Omron CX-Programmer project Karosszeria_gyartosor (CX-Programmer 9.10)

# PLC PLC: CJ2M CPU32
I/O table (CPU CJ2M-CPU32): rack 0 slot 0 CJ1W-ID211; rack 0 slot 1 CJ1W-OD212; rack 0 slot 2 CJ1W-ID211; rack 0 slot 3 CJ1W-OD212; rack 0 slot 11 CJ2M-EIP21

## Global symbols (name address type ; comment)
CRANE_Seq_1 D90 UINT[10]  ; Az 1-es típusú karosszéria átemelési feladatának pozícióit tartalmazó tömb.
CRANE_Seq_1_Lenght D41 UINT  ; Az 1-es típusú karosszéria átemelési feladatának pozícióit tartalmazó tömb hossza.
CRANE_Seq_2 D107 UINT[8]  ; Az 2-es típusú karosszéria átemelési feladatának pozícióit tartalmazó tömb.
CRANE_Seq_2_Lenght D75 UINT  ; Az 2-es típusú karosszéria átemelési feladatának pozícióit tartalmazó tömb hossza.
CRANE_Seq_3 D81 UINT[8]  ; Az 3-as típusú karosszéria átemelési feladatának pozícióit tartalmazó tömb.
CRANE_Seq_3_Lenght D76 UINT  ; Az 3-as típusú karosszéria átemelési feladatának pozícióit tartalmazó tömb hossza.
GRIPPER_CLOSE_POINT D123 UINT  ; A daru megfogójának zárását jelző index.
GRIPPER_OPEN_POINT D124 UINT  ; A daru megfogójának nyitását jelző index.
INPUT 2 UINT  ; A vezérlés bemenete.
IN_Acknowledgement 2.13 BOOL  ; Nyugtázás
IN_Body_Type_B0 2.00 BOOL  ; Utoljára beadott karosszéria típusa
IN_Body_Type_B1 2.01 BOOL  ; Utoljára beadott karosszéria típusa
IN_Emergency_Stop 2.14 BOOL  ; Vészstop
IN_Operator_Movement 2.08 BOOL  ; Operátor mozgása
IN_Robot_1_Done 2.09 BOOL  ; Robot 1 mozgás befejezve
IN_Robot_2_Done 2.10 BOOL  ; Robot 2 mozgás befejezve
IN_Robot_3_Done 2.11 BOOL  ; Festőrobot mozgás befejezve
IN_Sensor_Cell_1 2.05 BOOL  ; Cella 1
IN_Sensor_Cell_1_Arrival 2.02 BOOL  ; Cella 1 érkezés
IN_Sensor_Cell_2 2.06 BOOL  ; Cella 2
IN_Sensor_Cell_2_Arrival 2.03 BOOL  ; Cella 2 érkezés
IN_Sensor_Cell_3 2.07 BOOL  ; Cella 3
IN_Sensor_Cell_3_Arrival 2.04 BOOL  ; Cella 3 érkezés
IN_Unused 2.15 BOOL  ; Nincs használatban
IN_Warm_Reset 2.12 BOOL  ; Factory reset (warm reset)
OUTPUT 3 UINT  ; A vezérlés kimenete.
OUT_Belt_1_Switch 3.09 BOOL  ; Futószalag 1
OUT_Belt_2_Switch 3.10 BOOL  ; Futószalag 2
OUT_Belt_3_Switch 3.11 BOOL  ; Futószalag 3
OUT_Crane_Effector 3.15 BOOL  ; Daru megfogó vezérlése
OUT_Crane_Position_B0 3.12 BOOL  ; Daru pozíció
OUT_Crane_Position_B1 3.13 BOOL  ; Daru pozíció
OUT_Crane_Position_B2 3.14 BOOL  ; Daru pozíció
OUT_Robot_Effector 3.07 BOOL  ; Hegesztőpisztoly vagy a festékszóró vezérlése
OUT_Robot_Position_B0 3.04 BOOL  ; Robot adott konfiguráció vezérlése
OUT_Robot_Position_B1 3.05 BOOL  ; Robot adott konfiguráció vezérlése
OUT_Robot_Position_B2 3.06 BOOL  ; Robot adott konfiguráció vezérlése
OUT_Robot_Select_B0 3.00 BOOL  ; Robot kiválasztása
OUT_Robot_Select_B1 3.01 BOOL  ; Robot kiválasztása
OUT_Robot_Speed 3.02 BOOL  ; Robot lassú-gyors
OUT_Robot_Start 3.08 BOOL  ; Robotmozgás érvényesítés
OUT_Robot_Stop 3.03 BOOL  ; Robot állj
PAINTING_POINT_1 D80 UINT  ; Az első festési pont indexe.
PAINTING_POINT_2 D89 UINT  ; A második festési pont indexe.
ROBOT_Seq_1 D47 UINT[10]  ; Az 1-es típusú karosszérián elvégezendő hegesztési munkálatok pozícióit tartalmazó tömb.
ROBOT_Seq_1_Lenght D5 UINT  ; Az 1-es típusú karosszérián elvégezendő hegesztési munkálatok pozícióit tartalmazó tömb hossza
ROBOT_Seq_2 D57 UINT[10]  ; Az 2-es és 3-as típusú karosszériákon elvégezendő hegesztési munkálatok pozícióit tartalmazó tömb.
ROBOT_Seq_2_Lenght D19 UINT  ; Az 2-es és 3-as típusú karosszériákon elvégezendő hegesztési munkálatok pozícióit tartalmazó tömb hossza.
ROBOT_Seq_3 D35 UINT[5]  ; A karosszériákon elvégezendő festési munkálatok pozícióit tartalmazó tömb.
ROBOT_Seq_3_Lenght D40 UINT  ; A karosszériákon elvégezendő festési munkálatok pozícióit tartalmazó tömb hossza.
WELDING_POINT_1 D77 UINT  ; Az első hegesztési pont indexe.
WELDING_POINT_2 D78 UINT  ; A második hegesztési pont indexe.
WELDING_POINT_3 D79 UINT  ; A harmadik hegesztési pont indexe.

## Program Main (cyclic task 0)
Local symbols
BELT_ALL_State D17.00 BOOL[3]  ; A futószalagok állapotait tároló tömb.
CELL_1_BOOL_Array W10.00 BOOL[16]  ; Az első cella vezérlésénél az UINT típusok egyes bitjeinek eléréséhez használt tömb.
CELL_1_UINT_Value W10 UINT  ; Az első cella vezérlésénél az UINT típusok egyes bitjeinek eléréséhez használt változó.
CELL_2_BOOL_Array W20.00 BOOL[16]  ; A második cella vezérlésénél az UINT típusok egyes bitjeinek eléréséhez használt tömb.
CELL_2_UINT_Value W20 UINT  ; A második cella vezérlésénél az UINT típusok egyes bitjeinek eléréséhez használt változó.
CELL_3_BOOL_Array W30.00 BOOL[16]  ; A harmadik cella vezérlésénél az UINT típusok egyes bitjeinek eléréséhez használt tömb.
CELL_3_Crane_Startup D1.07 BOOL  ; A daru kezdeti állapotának beállítását jelző bit.
CELL_3_UINT_Value W30 UINT  ; A harmadik cella vezérlésénél az UINT típusok egyes bitjeinek eléréséhez használt változó.
CELL_ALL_Content D30 UINT[3]  ; A cellákban bent levő karosszériák típusszámai.
CELL_ALL_Speed_Bit D1.00 BOOL[3]  ; A cellákban dolgozó robotok sebességeit jelölő bitek tömbje.
CELL_ALL_Start_Bit D1.06 BOOL  ; A robotkonfigurációk kiadását és érvényesítését kölcsönösen kizáró jelzőbit.
CELL_ALL_Stop_Bit D17.04 BOOL[3]  ; A cellákban üzemelő munkagépek megállításának jelzőbitje.
CRANE_Gripper_Op D0.09 BOOL  ; A daru megfogójának állapotváltozását jelző bit.
CRANE_Highest_Seq_Index D8 UINT  ; A daru műveletsorának legmagasabb indexe.
CRANE_Op_Index D3 UINT  ; A daru aktuális műveletének indexe.
CV_Acknowledge_Needed D6.03 BOOL  ; A folytatáshoz nyugtázás szükségességét jelző bit.
CV_Belt_1_On D0.02 BOOL  ; A 1-es futószalag elindításának jelzőbitje.
CV_Belt_2_On D0.00 BOOL  ; A 2-es futószalag elindításának jelzőbitje.
CV_Belt_3_On D0.11 BOOL  ; A 3-es futószalag elindításának jelzőbitje.
CV_Crane_Finished D0.13 BOOL  ; A daru mozgásának befejeződését jelölő bit.
CV_Crane_Has_Next_Op D1.05 BOOL  ; A daru további műveleteit jelző bit.
CV_Crane_Op_Ended D1.04 BOOL  ; A daru további műveleteinek végét jelző bit.
CV_Crane_Ready D0.08 BOOL  ; A daru kezdeti pozíciójának felvételét jelző bit.
CV_Crane_Set_Operation D0.12 BOOL  ; A darut vezérlő kimenetek beállítását és a daru automatikus elindulását jelző bit.
CV_Delay_Ended D1.10 BOOL  ; A mintavételezés következő fázisa előtti késleltetés letelését jelző bit.
CV_Init_Done D0.10 BOOL  ; Az inicializáció befejeződését jelző bit.
CV_Preparation_Done D1.14 BOOL  ; A mintavételező alaphelyzetbe állításának jelzőbitje.
CV_Robot_1_2_Finished D0.03 BOOL  ; A 1-es és 2-es robotok mozgásának befejeződését jelölő bit.
CV_Robot_1_2_Has_Next_Op D0.04 BOOL  ; A 1-es és 2-es robotok további műveleteit jelző bit.
CV_Robot_1_2_Op_Ended D0.05 BOOL  ; A 1-es és 2-es robotok további műveleteinek végét jelző bit.
CV_Robot_1_2_Output_Set D0.06 BOOL  ; A 1-es és 2-es robotok esetén a kimenetek beállítását jelző bit.
CV_Robot_3_Finished D17.03 BOOL  ; A 3-as robot mozgásának befejeződését jelölő bit.
CV_Robot_3_Has_Next_Op D0.07 BOOL  ; A 3-as robot további műveleteit jelző bit.
CV_Robot_3_Op_Ended D1.03 BOOL  ; A 3-as robot további műveleteinek végét jelző bit.
CV_Robot_3_Output_Set D0.01 BOOL  ; A 3-as robot esetén a kimenetek beállítását jelző bit.
CV_Robot_All_Has_Next D17.11 BOOL  ; A robotok együttes vezérlése esetén további robotok sorban állását jelző bit.
CV_Robot_All_Output_Set D17.10 BOOL  ; A soron következő robot esetén a kimenetek beállítását jelző bit.
CV_Robot_All_Started D0.15 BOOL  ; A robot sikeres elindítását jelző bit.
CV_Robot_All_Update_Ended D17.12 BOOL  ; A robotok együttes vezérlése esetén a vezérlés befejezését jelző bit.
CV_Robots_Up_To_Date D6.05 BOOL  ; A robotkonfigurációk aktualitásának jelzőbitje.
CV_Robots_Update_Needed D6.04 BOOL  ; A robotkonfigurációk frissítési igényének jelzőbitje.
CV_Sample_Has_Next D1.12 BOOL  ; A minta beolvasásának következő lépését jelző bit.
CV_Sample_Read D1.11 BOOL  ; A minta beolvasását jelző bit.
CV_Signal_Read D1.09 BOOL  ; A minta következő bitjének beolvasását jelző bit.
CV_Startup_Done D1.08 BOOL  ; A szimuláció által kiküldött reset jel lefutását jelölő bit.
CV_Warm_Reset D0.14 BOOL  ; A szoftveres reset jelzőbitje.
Crane_TIMER T0002 TIMER  ; A darura mozgatásának befejeződésére várakoztató időzítő.
Gripper_TIMER T0001 TIMER  ; A darura szerelt megfogó nyitásának és zárásának befejeződésére várakoztató időzítő.
ROBOT_1_2_Highest_Seq_Index D9 UINT  ; Az 1-es és 2-es robotok műveletsorainak legmagasabb indexe.
ROBOT_1_2_Op_Index D2 UINT  ; Az 1-es és 2-es robotok aktuális műveletének indexe.
ROBOT_3_Op_Index D4 UINT  ; A 3-as robot aktuális műveletének indexe.
ROBOT_ALL_Delay T0003 TIMER  ; A robotok indítását követően a befejezés ellenőrzésének késleltetését szolgáló időzítő.
ROBOT_ALL_Effector_State D17.07 BOOL[3]  ; A robotok megmunkálóeszközeinek állapotai.
ROBOT_ALL_Index D33 UINT  ; A robotok egymás utáni vezérlésének indexe.
ROBOT_ALL_Position D125 UINT[3]  ; A robotok érvényes pozíciói.
SAFETY_Logical_HIGH D10 UINT  ; Az operátor mozgását jelző bemeneten mintavételezett magas logikai értékek száma.
SAFETY_Logical_LOW D11 UINT  ; Az operátor mozgását jelző bemeneten mintavételezett alacsony logikai értékek száma.
SAFETY_Operator_Position D18 UINT  ; Az operátor aktuális tartózkodási helye.
SAMPLER_Read_Index D16 UINT  ; A mintavételező indexsze.
Safety_BOOL_Array W40.00 BOOL[16]  ; A biztonsági intézkedéseknél az UINT típusok egyes bitjeinek eléréséhez használt tömb.
Safety_UINT_Value W40 UINT  ; A biztonsági intézkedéseknél az UINT típusok egyes bitjeinek eléréséhez használt változó.
Sampler_TIMER T0004 TIMER  ; A mintavételező késleltetését végző időzítő.
Selected_ROBOT D7 UINT  ; Az aktuálisan vezérelt robot indexe.
Start_HOLD T0000 TIMER  ; A robotpozíciókat érvényesítő bitet 1 másodpercig magas logikai szinten tartó időzítő.
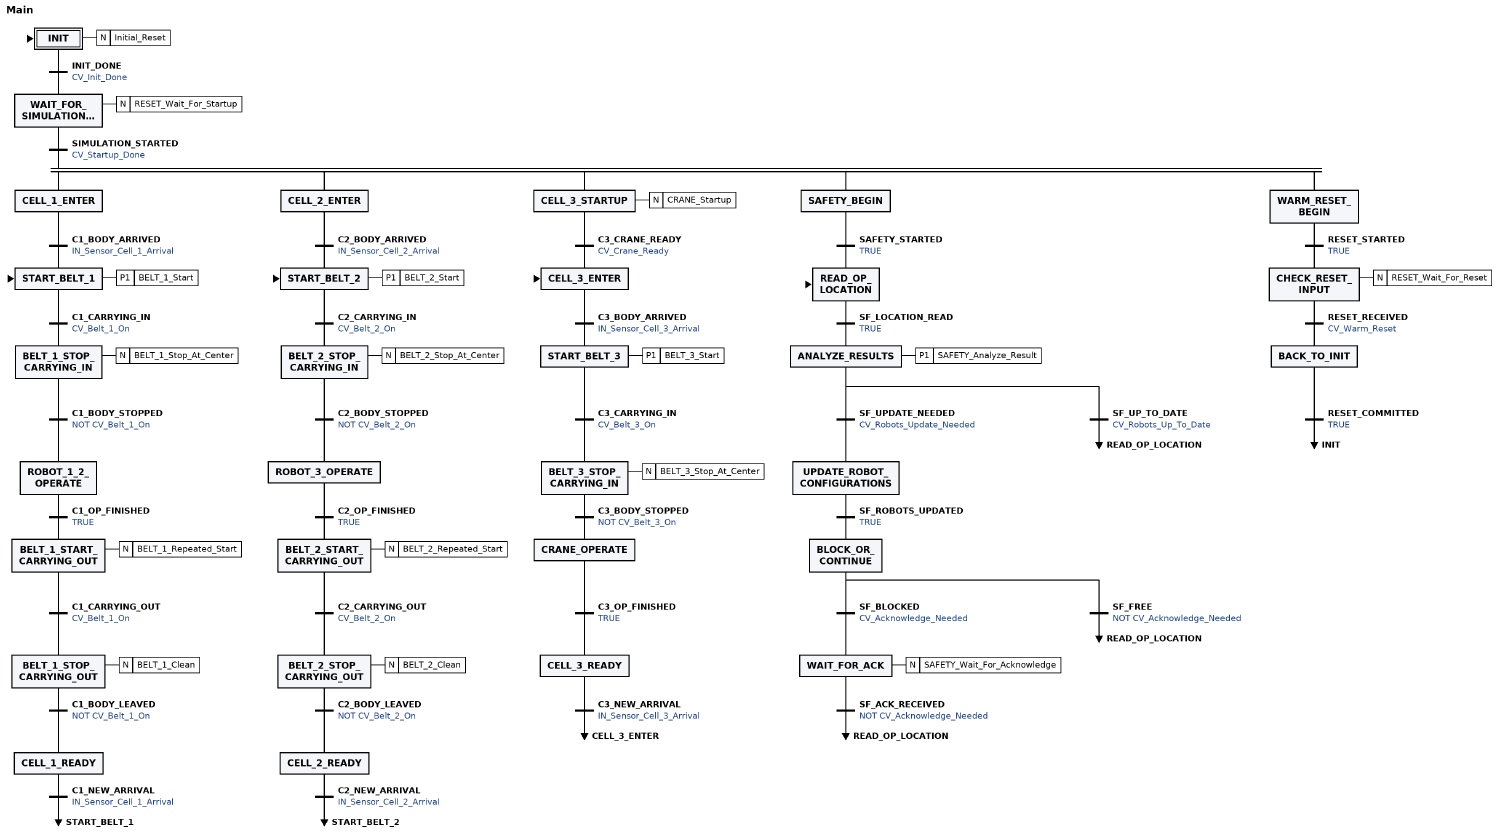
INITIAL_STEP INIT :
Initial_Reset(N) ;
END_STEP
TRANSITION INIT_DONE FROM INIT TO WAIT_FOR_SIMULATION_STARTUP
 := CV_Init_Done;
END_TRANSITION
STEP CELL_1_ENTER :
END_STEP
STEP CELL_2_ENTER :
END_STEP
STEP CELL_3_ENTER :
END_STEP
TRANSITION C1_BODY_ARRIVED FROM CELL_1_ENTER TO START_BELT_1
 := IN_Sensor_Cell_1_Arrival;
END_TRANSITION
STEP START_BELT_1 :
BELT_1_Start(P1) ;
END_STEP
TRANSITION C2_BODY_ARRIVED FROM CELL_2_ENTER TO START_BELT_2
 := IN_Sensor_Cell_2_Arrival;
END_TRANSITION
STEP START_BELT_2 :
BELT_2_Start(P1) ;
END_STEP
TRANSITION C2_CARRYING_IN FROM START_BELT_2 TO BELT_2_STOP_CARRYING_IN
 := CV_Belt_2_On;
END_TRANSITION
STEP BELT_2_STOP_CARRYING_IN :
BELT_2_Stop_At_Center(N) ;
END_STEP
TRANSITION C2_BODY_STOPPED FROM BELT_2_STOP_CARRYING_IN TO ROBOT_3_OPERATE
 := NOT CV_Belt_2_On;
END_TRANSITION
SUBCHART_STEP ROBOT_3_OPERATE :
Robot_3_Operation
END_STEP
TRANSITION C2_OP_FINISHED FROM ROBOT_3_OPERATE TO BELT_2_START_CARRYING_OUT
 := TRUE;
END_TRANSITION
STEP BELT_2_START_CARRYING_OUT :
BELT_2_Repeated_Start(N) ;
END_STEP
TRANSITION C2_CARRYING_OUT FROM BELT_2_START_CARRYING_OUT TO BELT_2_STOP_CARRYING_OUT
 := CV_Belt_2_On;
END_TRANSITION
STEP CELL_2_READY :
END_STEP
TRANSITION C2_NEW_ARRIVAL FROM CELL_2_READY TO START_BELT_2
 := IN_Sensor_Cell_2_Arrival;
END_TRANSITION
STEP BELT_2_STOP_CARRYING_OUT :
BELT_2_Clean(N) ;
END_STEP
TRANSITION C2_BODY_LEAVED FROM BELT_2_STOP_CARRYING_OUT TO CELL_2_READY
 := NOT CV_Belt_2_On;
END_TRANSITION
TRANSITION C1_CARRYING_IN FROM START_BELT_1 TO BELT_1_STOP_CARRYING_IN
 := CV_Belt_1_On;
END_TRANSITION
STEP BELT_1_STOP_CARRYING_IN :
BELT_1_Stop_At_Center(N) ;
END_STEP
TRANSITION C1_BODY_STOPPED FROM BELT_1_STOP_CARRYING_IN TO ROBOT_1_2_OPERATE
 := NOT CV_Belt_1_On;
END_TRANSITION
SUBCHART_STEP ROBOT_1_2_OPERATE :
Robot_1_2_Operation
END_STEP
TRANSITION C1_OP_FINISHED FROM ROBOT_1_2_OPERATE TO BELT_1_START_CARRYING_OUT
 := TRUE;
END_TRANSITION
STEP BELT_1_START_CARRYING_OUT :
BELT_1_Repeated_Start(N) ;
END_STEP
TRANSITION C1_CARRYING_OUT FROM BELT_1_START_CARRYING_OUT TO BELT_1_STOP_CARRYING_OUT
 := CV_Belt_1_On;
END_TRANSITION
STEP BELT_1_STOP_CARRYING_OUT :
BELT_1_Clean(N) ;
END_STEP
TRANSITION C1_BODY_LEAVED FROM BELT_1_STOP_CARRYING_OUT TO CELL_1_READY
 := NOT CV_Belt_1_On;
END_TRANSITION
STEP CELL_1_READY :
END_STEP
TRANSITION C1_NEW_ARRIVAL FROM CELL_1_READY TO START_BELT_1
 := IN_Sensor_Cell_1_Arrival;
END_TRANSITION
TRANSITION C3_BODY_ARRIVED FROM CELL_3_ENTER TO START_BELT_3
 := IN_Sensor_Cell_3_Arrival;
END_TRANSITION
STEP CELL_3_STARTUP :
CRANE_Startup(N) ;
END_STEP
TRANSITION C3_CRANE_READY FROM CELL_3_STARTUP TO CELL_3_ENTER
 := CV_Crane_Ready;
END_TRANSITION
STEP START_BELT_3 :
BELT_3_Start(P1) ;
END_STEP
TRANSITION C3_CARRYING_IN FROM START_BELT_3 TO BELT_3_STOP_CARRYING_IN
 := CV_Belt_3_On;
END_TRANSITION
STEP BELT_3_STOP_CARRYING_IN :
BELT_3_Stop_At_Center(N) ;
END_STEP
TRANSITION C3_BODY_STOPPED FROM BELT_3_STOP_CARRYING_IN TO CRANE_OPERATE
 := NOT CV_Belt_3_On;
END_TRANSITION
SUBCHART_STEP CRANE_OPERATE :
Crane_Operation
END_STEP
TRANSITION C3_OP_FINISHED FROM CRANE_OPERATE TO CELL_3_READY
 := TRUE;
END_TRANSITION
STEP CELL_3_READY :
END_STEP
TRANSITION C3_NEW_ARRIVAL FROM CELL_3_READY TO CELL_3_ENTER
 := IN_Sensor_Cell_3_Arrival;
END_TRANSITION
STEP SAFETY_BEGIN :
END_STEP
TRANSITION SAFETY_STARTED FROM SAFETY_BEGIN TO READ_OP_LOCATION
 := TRUE;
END_TRANSITION
STEP WAIT_FOR_SIMULATION_STARTUP :
RESET_Wait_For_Startup(N) ;
END_STEP
TRANSITION SIMULATION_STARTED FROM WAIT_FOR_SIMULATION_STARTUP TO (CELL_1_ENTER,CELL_2_ENTER,CELL_3_STARTUP,SAFETY_BEGIN,WARM_RESET_BEGIN)
 := CV_Startup_Done;
END_TRANSITION
SUBCHART_STEP READ_OP_LOCATION :
Safety_Get_Sample
END_STEP
TRANSITION SF_LOCATION_READ FROM READ_OP_LOCATION TO ANALYZE_RESULTS
 := TRUE;
END_TRANSITION
STEP ANALYZE_RESULTS :
SAFETY_Analyze_Result(P1) ;
END_STEP
SUBCHART_STEP UPDATE_ROBOT_CONFIGURATIONS :
Update_Robots
END_STEP
TRANSITION SF_ROBOTS_UPDATED FROM UPDATE_ROBOT_CONFIGURATIONS TO BLOCK_OR_CONTINUE
 := TRUE;
END_TRANSITION
STEP BLOCK_OR_CONTINUE :
END_STEP
TRANSITION SF_BLOCKED (PRIORITY := 1) FROM BLOCK_OR_CONTINUE TO WAIT_FOR_ACK
 := CV_Acknowledge_Needed;
END_TRANSITION
TRANSITION SF_FREE (PRIORITY := 2) FROM BLOCK_OR_CONTINUE TO READ_OP_LOCATION
 := NOT CV_Acknowledge_Needed;
END_TRANSITION
STEP WAIT_FOR_ACK :
SAFETY_Wait_For_Acknowledge(N) ;
END_STEP
TRANSITION SF_ACK_RECEIVED FROM WAIT_FOR_ACK TO READ_OP_LOCATION
 := NOT CV_Acknowledge_Needed;
END_TRANSITION
TRANSITION SF_UPDATE_NEEDED (PRIORITY := 1) FROM ANALYZE_RESULTS TO UPDATE_ROBOT_CONFIGURATIONS
 := CV_Robots_Update_Needed;
END_TRANSITION
TRANSITION SF_UP_TO_DATE (PRIORITY := 2) FROM ANALYZE_RESULTS TO READ_OP_LOCATION
 := CV_Robots_Up_To_Date;
END_TRANSITION
STEP WARM_RESET_BEGIN :
END_STEP
TRANSITION RESET_STARTED FROM WARM_RESET_BEGIN TO CHECK_RESET_INPUT
 := TRUE;
END_TRANSITION
STEP CHECK_RESET_INPUT :
RESET_Wait_For_Reset(N) ;
END_STEP
TRANSITION RESET_RECEIVED FROM CHECK_RESET_INPUT TO BACK_TO_INIT
 := CV_Warm_Reset;
END_TRANSITION
STEP BACK_TO_INIT :
END_STEP
TRANSITION RESET_COMMITTED FROM BACK_TO_INIT TO INIT
 := TRUE;
END_TRANSITION

### Action Initial_Reset
(* Kimenetek nullázása. *)
OUT_Robot_Select_B0	:= FALSE;
OUT_Robot_Select_B1	:= FALSE;
OUT_Robot_Speed		:= FALSE;
OUT_Robot_Stop		:= FALSE;
OUT_Robot_Position_B0	:= FALSE;
OUT_Robot_Position_B1	:= FALSE;
OUT_Robot_Position_B2	:= FALSE;
OUT_Robot_Effector	:= FALSE;
OUT_Robot_Start		:= FALSE;
OUT_Belt_1_Switch	:= FALSE;
OUT_Belt_2_Switch	:= FALSE;
OUT_Belt_3_Switch	:= FALSE;
OUT_Crane_Position_B0	:= FALSE;
OUT_Crane_Position_B1	:= FALSE;
OUT_Crane_Position_B2	:= FALSE;
OUT_Crane_Effector	:= FALSE;

(* Az előre meghatározott robotpozíciók beállítása. *)
ROBOT_Seq_1[0]	:= 5;
ROBOT_Seq_1[1]	:= 1;
ROBOT_Seq_1[2]	:= 5;
ROBOT_Seq_1[3]	:= 6;
ROBOT_Seq_1[4]	:= 2;
ROBOT_Seq_1[5]	:= 6;
ROBOT_Seq_1[6]	:= 7;
ROBOT_Seq_1[7]	:= 3;
ROBOT_Seq_1[8]	:= 7;
ROBOT_Seq_1[9]	:= 0;
ROBOT_Seq_1_Lenght	:= 10;

ROBOT_Seq_2[0]	:= 7;
ROBOT_Seq_2[1]	:= 3;
ROBOT_Seq_2[2]	:= 7;
ROBOT_Seq_2[3]	:= 6;
ROBOT_Seq_2[4]	:= 2;
ROBOT_Seq_2[5]	:= 6;
ROBOT_Seq_2[6]	:= 5;
ROBOT_Seq_2[7]	:= 1;
ROBOT_Seq_2[8]	:= 5;
ROBOT_Seq_2[9]	:= 0;
ROBOT_Seq_2_Lenght	:= 10;

ROBOT_Seq_3[0]	:= 1;
ROBOT_Seq_3[1]	:= 2;
ROBOT_Seq_3[2]	:= 3;
ROBOT_Seq_3[3]	:= 5;
ROBOT_Seq_3[4]	:= 0;
ROBOT_Seq_3_Lenght	:= 5;

(* Az előre meghatározott darupozíciók beállítása. *)
CRANE_Seq_1[0]	:= 0;
CRANE_Seq_1[1]	:= 0;
CRANE_Seq_1[2]	:= 1;
CRANE_Seq_1[3]	:= 3;
CRANE_Seq_1[4]	:= 5;
CRANE_Seq_1[5]	:= 4;
CRANE_Seq_1[6]	:= 4;
CRANE_Seq_1[7]	:= 5;
CRANE_Seq_1[8]	:= 3;
CRANE_Seq_1[9]	:= 1;
CRANE_Seq_1_Lenght	:= 10;

CRANE_Seq_2[0]	:= 0;
CRANE_Seq_2[1]	:= 0;
CRANE_Seq_2[2]	:= 1;
CRANE_Seq_2[3]	:= 3;
CRANE_Seq_2[4]	:= 2;
CRANE_Seq_2[5]	:= 2;
CRANE_Seq_2[6]	:= 3;
CRANE_Seq_2[7]	:= 1;
CRANE_Seq_2_Lenght	:= 8;

CRANE_Seq_3[0]	:= 0;
CRANE_Seq_3[1]	:= 0;
CRANE_Seq_3[2]	:= 1;
CRANE_Seq_3[3]	:= 7;
CRANE_Seq_3[4]	:= 6;
CRANE_Seq_3[5]	:= 6;
CRANE_Seq_3[6]	:= 7;
CRANE_Seq_3[7]	:= 1;
CRANE_Seq_3_Lenght	:= 8;

(* Az előre meghatározott állapotváltozások indexeinek beállítása. *)
WELDING_POINT_1	:= 1;
WELDING_POINT_2	:= 4;
WELDING_POINT_3	:= 7;
PAINTING_POINT_1	:= 1;
PAINTING_POINT_2	:= 2;
GRIPPER_CLOSE_POINT	:= 1;
GRIPPER_OPEN_POINT	:= 5;

(* Minden segédváltozó alaphelyzetbe állítása. *)
BELT_ALL_State[0]	:= FALSE;
BELT_ALL_State[1]	:= FALSE;
BELT_ALL_State[2]	:= FALSE;
CELL_1_UINT_Value	:= 0;
CELL_2_UINT_Value	:= 0;
CELL_3_Crane_Startup	:= FALSE;
CELL_3_UINT_Value	:= 0;
CELL_ALL_Content[0]	:= 0;
CELL_ALL_Content[1]	:= 0;
CELL_ALL_Content[2]	:= 0;
CELL_ALL_Speed_Bit[0]	:= FALSE;
CELL_ALL_Speed_Bit[1]	:= FALSE;
CELL_ALL_Speed_Bit[2]	:= FALSE;
CELL_ALL_Start_Bit	:= FALSE;
CELL_ALL_Stop_Bit[0]	:= FALSE;
CELL_ALL_Stop_Bit[1]	:= FALSE;
CELL_ALL_Stop_Bit[2]	:= FALSE;
CRANE_Gripper_Op	:= FALSE;
CRANE_Highest_Seq_Index	:= 0;
CRANE_Op_Index	:= 0;
CV_Acknowledge_Needed	:= FALSE;
CV_Belt_1_On	:= FALSE;
CV_Belt_2_On	:= FALSE;
CV_Belt_3_On	:= FALSE;
CV_Crane_Finished	:= FALSE;
CV_Crane_Has_Next_Op	:= FALSE;
CV_Crane_Op_Ended	:= FALSE;
CV_Crane_Ready	:= FALSE;
CV_Crane_Set_Operation	:= FALSE;
CV_Delay_Ended	:= FALSE;
CV_Init_Done	:= FALSE;
CV_Preparation_Done	:= FALSE;
CV_Robot_1_2_Finished	:= FALSE;
CV_Robot_1_2_Has_Next_Op	:= FALSE;
CV_Robot_1_2_Op_Ended	:= FALSE;
CV_Robot_1_2_Output_Set	:= FALSE;
CV_Robot_3_Finished	:= FALSE;
CV_Robot_3_Has_Next_Op	:= FALSE;
CV_Robot_3_Op_Ended	:= FALSE;
CV_Robot_3_Output_Set	:= FALSE;
CV_Robot_All_Has_Next	:= FALSE;
CV_Robot_All_Output_Set	:= FALSE;
CV_Robot_All_Started	:= FALSE;
CV_Robot_All_Update_Ended	:= FALSE;
CV_Robots_Up_To_Date	:= FALSE;
CV_Robots_Update_Needed	:= FALSE;
CV_Sample_Has_Next	:= FALSE;
CV_Sample_Read	:= FALSE;
CV_Signal_Read	:= FALSE;
CV_Startup_Done	:= FALSE;
CV_Warm_Reset	:= FALSE;
ROBOT_1_2_Highest_Seq_Index	:= 0;
ROBOT_1_2_Op_Index	:= 0;
ROBOT_3_Op_Index	:= 0;
ROBOT_ALL_Effector_State[0]	:= FALSE;
ROBOT_ALL_Effector_State[1]	:= FALSE;
ROBOT_ALL_Effector_State[2]	:= FALSE;
ROBOT_ALL_Index	:= 0;
ROBOT_ALL_Position[0]	:= 0;
ROBOT_ALL_Position[1]	:= 0;
ROBOT_ALL_Position[2]	:= 0;
SAFETY_Logical_HIGH	:= 0;
SAFETY_Logical_LOW	:= 0;
SAFETY_Operator_Position	:= 0;
Safety_UINT_Value	:= 0;
SAMPLER_Read_Index	:= 0;
Selected_ROBOT	:= 0;

(* Az inicializálció befejezésének jelzése. *)
CV_Init_Done := TRUE;

### Action BELT_1_Start
(* A karosszéria típust jelző bemenetek szerinti érték rögzítése. *)
CELL_1_UINT_Value := 0;
CELL_1_BOOL_Array[0] := IN_Body_Type_B0;
CELL_1_BOOL_Array[1] := IN_Body_Type_B1;
CELL_ALL_Content[0] := CELL_1_UINT_Value;

(* A cella futószalagjának bekapcsolása és az átmenet tüzelése. *)
OUT_Belt_1_Switch := TRUE;
CV_Belt_1_On := TRUE;

### Action BELT_1_Stop_At_Center

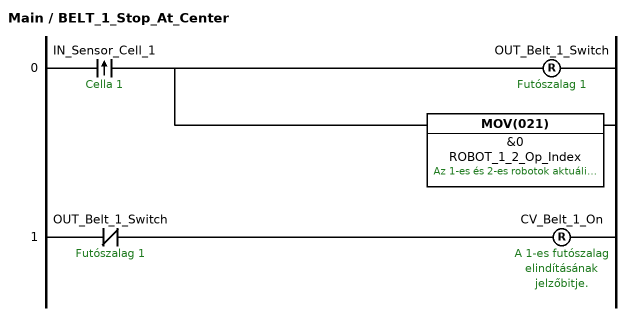
; rung 0
@LD IN_Sensor_Cell_1  ; Cella 1
RSET OUT_Belt_1_Switch  ; Futószalag 1
MOV(021) &0 ROBOT_1_2_Op_Index  ; Az 1-es és 2-es robotok aktuális műveletének indexe.
; rung 1
LDNOT OUT_Belt_1_Switch  ; Futószalag 1
RSET CV_Belt_1_On  ; A 1-es futószalag elindításának jelzőbitje.

### Action BELT_1_Repeated_Start
(* A cella futószalagjának bekapcsolása és az átmenet tüzelése, ha a soron következő cella üres. *)
IF CELL_ALL_Content[1] = 0 THEN
	OUT_Belt_1_Switch := TRUE;
	CV_Belt_1_On := TRUE;
END_IF;

### Action BELT_1_Clean

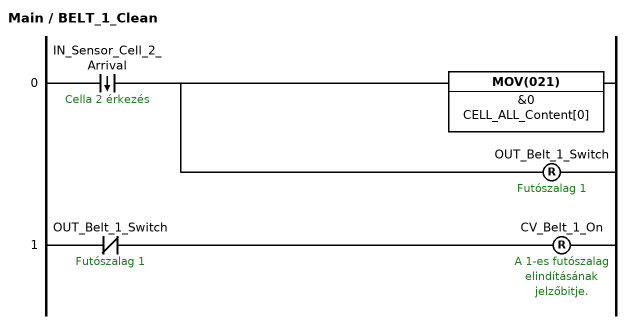
; rung 0
%LD IN_Sensor_Cell_2_Arrival  ; Cella 2 érkezés
MOV(021) &0 CELL_ALL_Content[0]
RSET OUT_Belt_1_Switch  ; Futószalag 1
; rung 1
LDNOT OUT_Belt_1_Switch  ; Futószalag 1
RSET CV_Belt_1_On  ; A 1-es futószalag elindításának jelzőbitje.

### Action BELT_2_Start
(* Az előző cellában rögzített karosszéria típus átmásolása, ha az előző cella futószalagja mozgásban van, *)
(* egyébként a karosszéria típust jelző bemenetek szerinti érték rögzítése. *)
IF OUT_Belt_1_Switch = TRUE THEN
	CELL_ALL_Content[1] := CELL_ALL_Content[0];
ELSIF OUT_Belt_1_Switch = FALSE THEN
	CELL_2_UINT_Value := 0;
	CELL_2_BOOL_Array[0] := IN_Body_Type_B0;
	CELL_2_BOOL_Array[1] := IN_Body_Type_B1;
	CELL_ALL_Content[1] := CELL_2_UINT_Value;
END_IF;

(* A cella futószalagjának bekapcsolása és az átmenet tüzelése. *)
OUT_Belt_2_Switch := TRUE;
CV_Belt_2_On := TRUE;

### Action BELT_2_Stop_At_Center

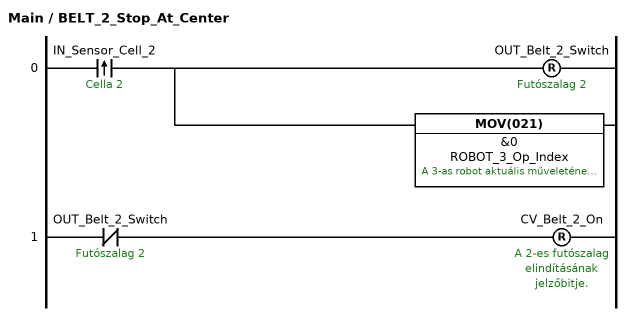
; rung 0
@LD IN_Sensor_Cell_2  ; Cella 2
RSET OUT_Belt_2_Switch  ; Futószalag 2
MOV(021) &0 ROBOT_3_Op_Index  ; A 3-as robot aktuális műveletének indexe.
; rung 1
LDNOT OUT_Belt_2_Switch  ; Futószalag 2
RSET CV_Belt_2_On  ; A 2-es futószalag elindításának jelzőbitje.

### Action BELT_2_Repeated_Start
(* A cella futószalagjának bekapcsolása és az átmenet tüzelése, ha a soron következő cella üres. *)
IF CELL_ALL_Content[2] = 0 THEN
	OUT_Belt_2_Switch := TRUE;
	CV_Belt_2_On := TRUE;
END_IF;

### Action BELT_2_Clean

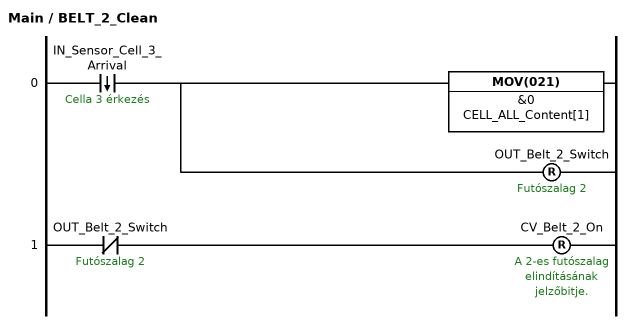
; rung 0
%LD IN_Sensor_Cell_3_Arrival  ; Cella 3 érkezés
MOV(021) &0 CELL_ALL_Content[1]
RSET OUT_Belt_2_Switch  ; Futószalag 2
; rung 1
LDNOT OUT_Belt_2_Switch  ; Futószalag 2
RSET CV_Belt_2_On  ; A 2-es futószalag elindításának jelzőbitje.

### Action BELT_3_Start
(* Az előző cellában rögzített karosszéria típus átmásolása, ha az előző cella futószalagja mozgásban van, *)
(* egyébként a karosszéria típust jelző bemenetek szerinti érték rögzítése. *)
IF OUT_Belt_2_Switch = TRUE THEN
	CELL_ALL_Content[2] := CELL_ALL_Content[1];
ELSIF OUT_Belt_2_Switch = FALSE THEN
	CELL_3_UINT_Value := 0;
	CELL_3_BOOL_Array[0] := IN_Body_Type_B0;
	CELL_3_BOOL_Array[1] := IN_Body_Type_B1;
	CELL_ALL_Content[2] := CELL_3_UINT_Value;
END_IF;

(* A cella futószalagjának bekapcsolása és az átmenet tüzelése. *)
OUT_Belt_3_Switch := TRUE;
CV_Belt_3_On := TRUE;

### Action BELT_3_Stop_At_Center

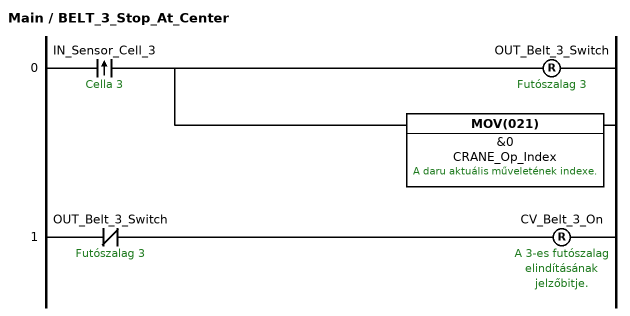
; rung 0
@LD IN_Sensor_Cell_3  ; Cella 3
RSET OUT_Belt_3_Switch  ; Futószalag 3
MOV(021) &0 CRANE_Op_Index  ; A daru aktuális műveletének indexe.
; rung 1
LDNOT OUT_Belt_3_Switch  ; Futószalag 3
RSET CV_Belt_3_On  ; A 3-es futószalag elindításának jelzőbitje.

### Action ROBOT_ALL_Set_Output
(* A robotok vezérléséhez tartoró kritikus szekció lezárása és a kimenetek beállítása, ha a kritikus szekció szabad. *)
IF CELL_ALL_Start_Bit = FALSE THEN
	CELL_ALL_Start_Bit := TRUE;

	(* A soron következő robot kiválasztása. *)
	Safety_UINT_Value := ROBOT_ALL_Index + 1;
	OUT_Robot_Select_B0 := Safety_BOOL_Array[0];
	OUT_Robot_Select_B1 := Safety_BOOL_Array[1];

	(* A soron következő robot érvényes pozíciójának beállítása a kimeneteken. *)
	Safety_UINT_Value := ROBOT_ALL_Position[ROBOT_ALL_Index];
	OUT_Robot_Position_B0 := Safety_BOOL_Array[0];
	OUT_Robot_Position_B1 := Safety_BOOL_Array[1];
	OUT_Robot_Position_B2 := Safety_BOOL_Array[2];

	(* A soron következő robot sebességeit befolyásoló kimenetek beállítása. *)
	IF ROBOT_ALL_Index < 2 THEN
		Safety_UINT_Value := 0;
	ELSE
		Safety_UINT_Value := 1;
	END_IF;
	OUT_Robot_Stop := CELL_ALL_Stop_Bit[Safety_UINT_Value];
	OUT_Robot_Speed := CELL_ALL_Speed_Bit[Safety_UINT_Value];

	(* A soron következő robot megmunkálókészülékének kikapcsolása leállítás esetén, *)
	(* ellenkező esetben az érvényes érték beállítása a kimeneten. *)
	IF CELL_ALL_Stop_Bit[Safety_UINT_Value] = TRUE THEN
		OUT_Robot_Effector := FALSE;
	ELSE
		OUT_Robot_Effector := ROBOT_ALL_Effector_State[ROBOT_ALL_Index];
	END_IF;

	(* A műveletsor későbbi átmeneteinek alaphelyzetbe állítása és a jelenlegi átmenet tüzelése. *)
	CV_Robot_All_Output_Set := FALSE;
	CV_Robot_All_Started := FALSE;
	CV_Robot_All_Has_Next := FALSE;
	CV_Robot_All_Update_Ended := FALSE;
	CV_Robot_All_Output_Set := TRUE;
END_IF;

### Action ROBOT_ALL_Start

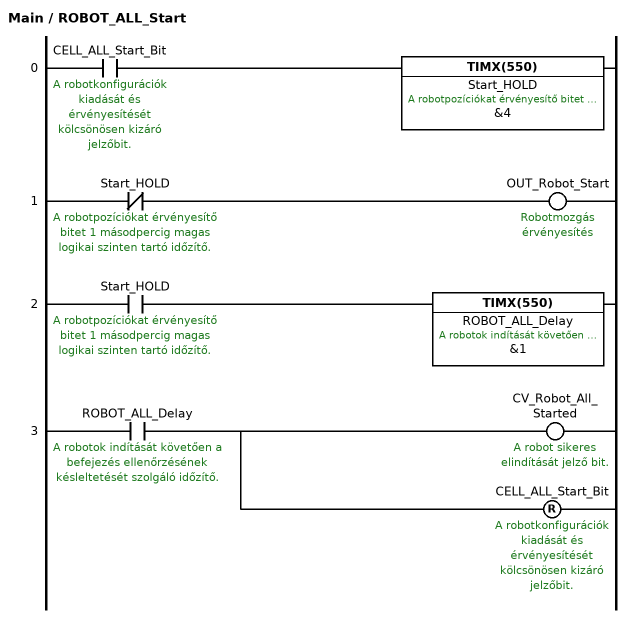
; rung 0
LD CELL_ALL_Start_Bit  ; A robotkonfigurációk kiadását és érvényesítését kölcsönösen kizáró jelzőbit.
TIMX(550) Start_HOLD &4  ; A robotpozíciókat érvényesítő bitet 1 másodpercig magas logikai szinten tartó időzítő.
; rung 1
LDNOT Start_HOLD  ; A robotpozíciókat érvényesítő bitet 1 másodpercig magas logikai szinten tartó időzítő.
OUT OUT_Robot_Start  ; Robotmozgás érvényesítés
; rung 2
LD Start_HOLD  ; A robotpozíciókat érvényesítő bitet 1 másodpercig magas logikai szinten tartó időzítő.
TIMX(550) ROBOT_ALL_Delay &1  ; A robotok indítását követően a befejezés ellenőrzésének késleltetését szolgáló időzítő.
; rung 3
LD ROBOT_ALL_Delay  ; A robotok indítását követően a befejezés ellenőrzésének késleltetését szolgáló időzítő.
OUT CV_Robot_All_Started  ; A robot sikeres elindítását jelző bit.
RSET CELL_ALL_Start_Bit  ; A robotkonfigurációk kiadását és érvényesítését kölcsönösen kizáró jelzőbit.

### Action ROBOT_ALL_Next_Step
(* A műveletsor befejezése, amennyiben az utolsó robot állapota is módosítva lett, *)
(* elllenkező esetben a soron következő robot indexének beállítása. *)
IF ROBOT_ALL_Index = 2 THEN
	ROBOT_ALL_Index := 0;
	CV_Robot_All_Has_Next := FALSE;
	CV_Robot_All_Update_Ended := TRUE;
ELSIF ROBOT_ALL_Index < 2 THEN
	ROBOT_ALL_Index := ROBOT_ALL_Index + 1;
	CV_Robot_All_Update_Ended := FALSE;
	CV_Robot_All_Has_Next := TRUE;
END_IF;

(* A kimenetek beállítását jelző bit törlése. *)
CV_Robot_All_Output_Set := FALSE;

### Action ROBOT_1_2_Set_Output
(* A robotok vezérléséhez tartoró kritikus szekció lezárása és a kimenetek beállítása, ha a kritikus szekció szabad. *)
IF CELL_ALL_Start_Bit = FALSE THEN
	CELL_ALL_Start_Bit := TRUE;

	(* Az 1-es robot kiválasztása, amennyiben a cellában levő karosszéria típusa 1-es, *)
	(* egyébkén a 2-es robot kiválasztása. *)
	IF CELL_ALL_Content[0] = 1 THEN
		OUT_Robot_Select_B0 := TRUE;
		OUT_Robot_Select_B1 := FALSE;
		Selected_ROBOT := 0;
	ELSE
		OUT_Robot_Select_B0 := FALSE;
		OUT_Robot_Select_B1 := TRUE;
		Selected_ROBOT := 1;
	END_IF;
	
	(* A soron következő robotpozíciók beállítása a kimeneteken a karosszéria típusától függően. *)
	IF CELL_ALL_Content[0] = 1 THEN
		CELL_1_UINT_Value := ROBOT_Seq_1[ROBOT_1_2_Op_Index];
		ROBOT_1_2_Highest_Seq_Index := ROBOT_Seq_1_Lenght - 1;
	ELSE
		CELL_1_UINT_Value := ROBOT_Seq_2[ROBOT_1_2_Op_Index];
		ROBOT_1_2_Highest_Seq_Index := ROBOT_Seq_2_Lenght - 1;
	END_IF;
	OUT_Robot_Position_B0 := CELL_1_BOOL_Array[0];
	OUT_Robot_Position_B1 := CELL_1_BOOL_Array[1];
	OUT_Robot_Position_B2 := CELL_1_BOOL_Array[2];
	ROBOT_ALL_Position[Selected_ROBOT] := CELL_1_UINT_Value;

	(* A robot sebességeit befolyásoló kimenetek beállítása. *)
	OUT_Robot_Stop := CELL_ALL_Stop_Bit[0];
	OUT_Robot_Speed := CELL_ALL_Speed_Bit[0];

	(* A robot hegesztőkészülékének bekapcsolása a megfelelő pozíciókon. *)
	IF ROBOT_1_2_Op_Index = WELDING_POINT_1 OR ROBOT_1_2_Op_Index = WELDING_POINT_2 OR ROBOT_1_2_Op_Index = WELDING_POINT_3  THEN
		OUT_Robot_Effector := TRUE;
	ELSE
		OUT_Robot_Effector := FALSE;
	END_IF;
	ROBOT_ALL_Effector_State[Selected_ROBOT] := OUT_Robot_Effector;

	(* A műveletsor későbbi átmeneteinek alaphelyzetbe állítása és a jelenlegi átmenet tüzelése. *)
	CV_Robot_All_Started := FALSE;
	CV_Robot_1_2_Finished := FALSE;
	CV_Robot_1_2_Has_Next_Op := FALSE;
	CV_Robot_1_2_Op_Ended := FALSE;
	CV_Robot_1_2_Output_Set := TRUE;
END_IF;

### Action ROBOT_1_2_Wait_To_Finish

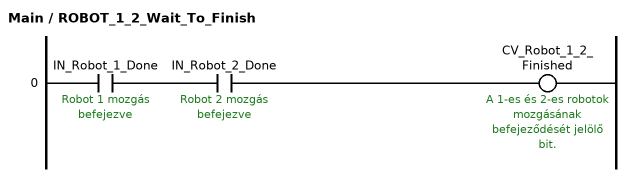
; rung 0
LD IN_Robot_1_Done  ; Robot 1 mozgás befejezve
AND IN_Robot_2_Done  ; Robot 2 mozgás befejezve
OUT CV_Robot_1_2_Finished  ; A 1-es és 2-es robotok mozgásának befejeződését jelölő bit.

### Action ROBOT_1_2_Next_Step
(* A műveletsor befejezése, amennyiben a robot az utolsó műveletet is elvégezte, ellenkező esetben a soron következő művelet indexének beállítása. *)
IF ROBOT_1_2_Op_Index = ROBOT_1_2_Highest_Seq_Index THEN
	ROBOT_1_2_Op_Index := 0;
	CV_Robot_1_2_Has_Next_Op := FALSE;
	CV_Robot_1_2_Op_Ended := TRUE;
ELSIF ROBOT_1_2_Op_Index < ROBOT_1_2_Highest_Seq_Index  THEN
	ROBOT_1_2_Op_Index := ROBOT_1_2_Op_Index + 1;
	CV_Robot_1_2_Op_Ended := FALSE;
	CV_Robot_1_2_Has_Next_Op := TRUE;
END_IF;

(* A kimenetek beállítását jelző bit törlése. *)
CV_Robot_1_2_Output_Set := FALSE;

### Action ROBOT_3_Set_Output
(* A robotok vezérléséhez tartoró kritikus szekció lezárása és a kimenetek beállítása, ha a kritikus szekció szabad. *)
IF CELL_ALL_Start_Bit = FALSE THEN
	CELL_ALL_Start_Bit := TRUE;

	(* A 3-as robot kiválasztása. *)
	OUT_Robot_Select_B0 := TRUE;
	OUT_Robot_Select_B1 := TRUE;
	Selected_ROBOT := 2;
	
	(* A soron következő robotpozíciók beállítása a kimeneteken. *)
	CELL_2_UINT_Value := ROBOT_Seq_3[ROBOT_3_Op_Index];
	OUT_Robot_Position_B0 := CELL_2_BOOL_Array[0];
	OUT_Robot_Position_B1 := CELL_2_BOOL_Array[1];
	OUT_Robot_Position_B2 := CELL_2_BOOL_Array[2];
	ROBOT_ALL_Position[Selected_ROBOT] := CELL_2_UINT_Value;


	(* A robot sebességeit befolyásoló kimenetek beállítása. *)
	OUT_Robot_Stop := CELL_ALL_Stop_Bit[1];
	OUT_Robot_Speed := CELL_ALL_Speed_Bit[1];

	(* A robot festőkészülékének bekapcsolása a megfelelő pozíciókon. *)
	IF ROBOT_3_Op_Index = PAINTING_POINT_1 OR ROBOT_3_Op_Index = PAINTING_POINT_2 THEN
		OUT_Robot_Effector := TRUE;
	ELSE
		OUT_Robot_Effector := FALSE;
	END_IF;
	ROBOT_ALL_Effector_State[Selected_ROBOT] := OUT_Robot_Effector;


	(* A műveletsor későbbi átmeneteinek alaphelyzetbe állítása és a jelenlegi átmenet tüzelése. *)
	CV_Robot_All_Started := FALSE;
	CV_Robot_3_Finished := FALSE;
	CV_Robot_3_Has_Next_Op := FALSE;
	CV_Robot_3_Op_Ended := FALSE;
	CV_Robot_3_Output_Set := TRUE;
END_IF;

### Action ROBOT_3_Wait_To_Finish

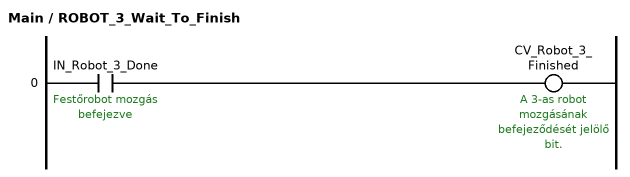
; rung 0
LD IN_Robot_3_Done  ; Festőrobot mozgás befejezve
OUT CV_Robot_3_Finished  ; A 3-as robot mozgásának befejeződését jelölő bit.

### Action ROBOT_3_Next_Step
(* A műveletsor befejezése, amennyiben a robot az utolsó műveletet is elvégezte, ellenkező esetben a soron következő művelet indexének beállítása. *)
IF ROBOT_3_Op_Index = (ROBOT_Seq_3_Lenght - 1) THEN
	ROBOT_3_Op_Index := 0;
	CV_Robot_3_Has_Next_Op := FALSE;
	CV_Robot_3_Op_Ended := TRUE;
ELSIF ROBOT_3_Op_Index <  (ROBOT_Seq_3_Lenght - 1) THEN
	ROBOT_3_Op_Index := ROBOT_3_Op_Index + 1;
	CV_Robot_3_Op_Ended := FALSE;
	CV_Robot_3_Has_Next_Op := TRUE;
END_IF;

(* A kimenetek beállítását jelző bit törlése. *)
CV_Robot_3_Output_Set := FALSE;

### Action CRANE_Startup

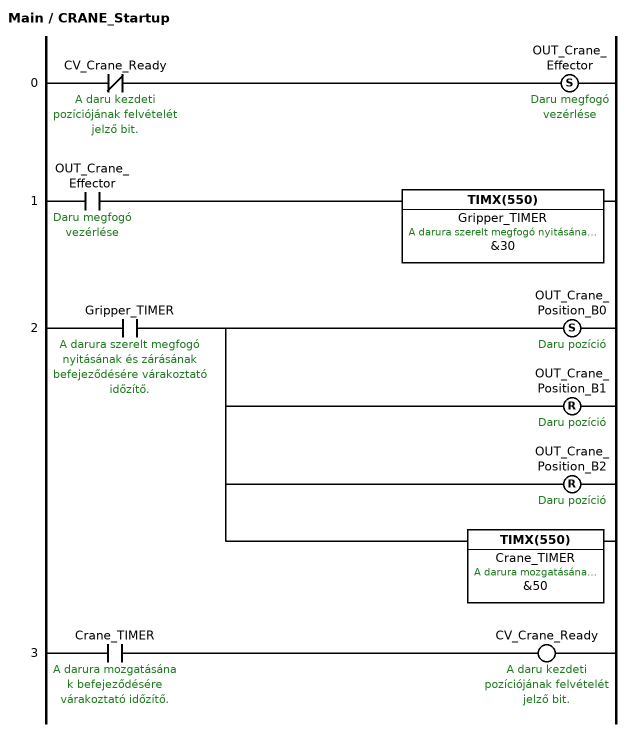
; rung 0
LDNOT CV_Crane_Ready  ; A daru kezdeti pozíciójának felvételét jelző bit.
SET OUT_Crane_Effector  ; Daru megfogó vezérlése
; rung 1
LD OUT_Crane_Effector  ; Daru megfogó vezérlése
TIMX(550) Gripper_TIMER &30  ; A darura szerelt megfogó nyitásának és zárásának befejeződésére várakoztató időzítő.
; rung 2
LD Gripper_TIMER  ; A darura szerelt megfogó nyitásának és zárásának befejeződésére várakoztató időzítő.
SET OUT_Crane_Position_B0  ; Daru pozíció
RSET OUT_Crane_Position_B1  ; Daru pozíció
RSET OUT_Crane_Position_B2  ; Daru pozíció
TIMX(550) Crane_TIMER &50  ; A darura mozgatásának befejeződésére várakoztató időzítő.
; rung 3
LD Crane_TIMER  ; A darura mozgatásának befejeződésére várakoztató időzítő.
OUT CV_Crane_Ready  ; A daru kezdeti pozíciójának felvételét jelző bit.

### Action CRANE_Set_Operation
(* A daru következő műveletének beállítása, amennyiben a vész-stop nem aktív. *)
IF CELL_ALL_Stop_Bit[2] = FALSE THEN
	(* A soron következő robotpozíciók beállítása a kimeneteken a karosszéria típusától függően. *)
	CASE CELL_ALL_Content[2] OF
		1:
			CELL_3_UINT_Value := CRANE_Seq_1[CRANE_Op_Index];
			CRANE_Highest_Seq_Index := CRANE_Seq_1_Lenght - 1;
			GRIPPER_OPEN_POINT := 6;
		2:
			CELL_3_UINT_Value := CRANE_Seq_2[CRANE_Op_Index];
			CRANE_Highest_Seq_Index := CRANE_Seq_2_Lenght - 1;
			GRIPPER_OPEN_POINT := 5;
		3:
			CELL_3_UINT_Value := CRANE_Seq_3[CRANE_Op_Index];
			CRANE_Highest_Seq_Index := CRANE_Seq_3_Lenght - 1;
			GRIPPER_OPEN_POINT := 5;
	END_CASE;
	OUT_Crane_Position_B0 := CELL_3_BOOL_Array[0];
	OUT_Crane_Position_B1 := CELL_3_BOOL_Array[1];
	OUT_Crane_Position_B2 := CELL_3_BOOL_Array[2];

	(* A daru megfogójának zárása a megfelelő pozíciókon. *)
	IF CRANE_Op_Index >= GRIPPER_CLOSE_POINT AND CRANE_Op_Index < GRIPPER_OPEN_POINT THEN
		OUT_Crane_Effector := FALSE;
	ELSE
		OUT_Crane_Effector := TRUE;
	END_IF;

	(* A daru megfogójának állapotváltozását jelző bit magas logikai szintre állítása, ha a megfogó állapota meg fog változni. *)
	IF CRANE_Op_Index = GRIPPER_CLOSE_POINT OR CRANE_Op_Index = GRIPPER_OPEN_POINT THEN
		CRANE_Gripper_Op := TRUE;
	ELSE
		CRANE_Gripper_Op := FALSE;
	END_IF;

	(* A műveletsor későbbi átmeneteinek alaphelyzetbe állítása és a jelenlegi átmenet tüzelése. *)
	CV_Crane_Finished := FALSE;
	CV_Crane_Has_Next_Op := FALSE;
	CV_Crane_Op_Ended := FALSE;
	CV_Crane_Set_Operation := TRUE;
END_IF;

### Action CRANE_Wait_To_Finish

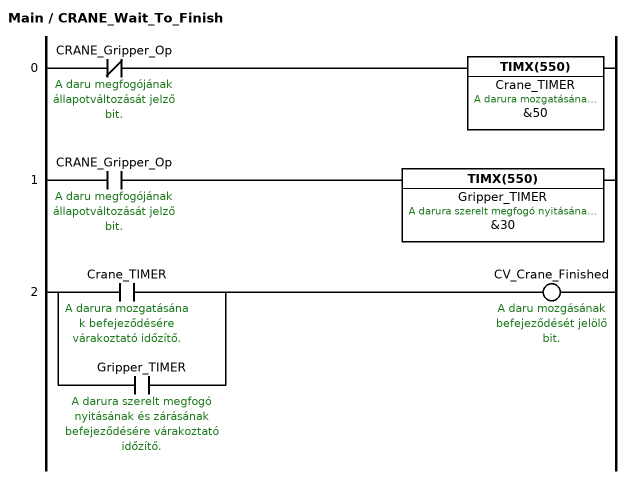
; rung 0
LDNOT CRANE_Gripper_Op  ; A daru megfogójának állapotváltozását jelző bit.
TIMX(550) Crane_TIMER &50  ; A darura mozgatásának befejeződésére várakoztató időzítő.
; rung 1
LD CRANE_Gripper_Op  ; A daru megfogójának állapotváltozását jelző bit.
TIMX(550) Gripper_TIMER &30  ; A darura szerelt megfogó nyitásának és zárásának befejeződésére várakoztató időzítő.
; rung 2
LD Crane_TIMER  ; A darura mozgatásának befejeződésére várakoztató időzítő.
OR Gripper_TIMER  ; A darura szerelt megfogó nyitásának és zárásának befejeződésére várakoztató időzítő.
OUT CV_Crane_Finished  ; A daru mozgásának befejeződését jelölő bit.

### Action CRANE_Next_Step
(* A műveletsor befejezése, amennyiben a daru az utolsó műveletet is elvégezte, ellenkező esetben a soron következő művelet indexének beállítása. *)
IF CRANE_Op_Index = CRANE_Highest_Seq_Index THEN
	CRANE_Op_Index := 0;
	CV_Crane_Has_Next_Op := FALSE;
	CV_Crane_Op_Ended := TRUE;
	CELL_ALL_Content[2]	:= 0;
ELSIF CRANE_Op_Index < CRANE_Highest_Seq_Index  THEN
	CRANE_Op_Index := CRANE_Op_Index + 1;
	CV_Crane_Op_Ended := FALSE;
	CV_Crane_Has_Next_Op := TRUE;
END_IF;

(* A kimenetek beállítását jelző bit törlése. *)
CV_Crane_Set_Operation := FALSE;

### Action SAMPLER_Reset_Sampler
(* Az operátor mozgását jelző bemenet egymásodperces állapotváltozását összegző regiszterek ürítése. *)
SAFETY_Logical_HIGH := 0;
SAFETY_Logical_LOW := 0;
SAMPLER_Read_Index := 0;
CV_Robots_Update_Needed := FALSE;
CV_Robots_Up_To_Date := FALSE;
CV_Preparation_Done := TRUE;

### Action SAMPLER_Read_Signal
(* Az operátor mozgását jelző bemenet aktuális értékének megfelelő regiszter növelése. *)
IF IN_Operator_Movement = TRUE THEN
	SAFETY_Logical_HIGH := SAFETY_Logical_HIGH + 1;
ELSE
	SAFETY_Logical_LOW := SAFETY_Logical_LOW + 1;
END_IF;
CV_Signal_Read := TRUE;

### Action SAMPLER_Read_Delay

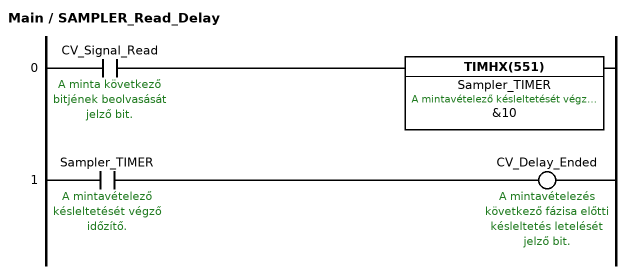
; rung 0
LD CV_Signal_Read  ; A minta következő bitjének beolvasását jelző bit.
TIMHX(551) Sampler_TIMER &10  ; A mintavételező késleltetését végző időzítő.
; rung 1
LD Sampler_TIMER  ; A mintavételező késleltetését végző időzítő.
OUT CV_Delay_Ended  ; A mintavételezés következő fázisa előtti késleltetés letelését jelző bit.

### Action SAMPLER_Next_Step
(* A műveletsor befejezése, amennyiben a mintavételező utolsó jelet is beolvasta, vagy a vész-stop be lett nyomva *)
(* ellenkező esetben az index növelése és a mintavételezés folytatása. *)
IF SAMPLER_Read_Index = 10 OR IN_Emergency_Stop = FALSE THEN
	SAMPLER_Read_Index := 0;
	CV_Sample_Has_Next := FALSE;
	CV_Sample_Read := TRUE;
ELSIF SAMPLER_Read_Index < 10 THEN
	SAMPLER_Read_Index := SAMPLER_Read_Index + 1;
	CV_Sample_Read := FALSE;
	CV_Sample_Has_Next := TRUE;
END_IF;

(* A mintavételezés segédbitjeinek törlése. *)
CV_Preparation_Done := FALSE;
CV_Signal_Read := FALSE;
CV_Delay_Ended := FALSE;

	

### Action SAFETY_Analyze_Result
(* Minden robot megállítása, ha a vész-stop meg lett nyomva. *)
IF IN_Emergency_Stop = FALSE THEN
	SAFETY_Operator_Position := 0;
	
	(* A robotkonfigurációk frissítésének és nyugtázás szükségességének jelzése. *)
	CV_Robots_Update_Needed := TRUE;
	CV_Robots_Up_To_Date := FALSE;
	CV_Acknowledge_Needed := TRUE;
	
	(* Minden cella stop bitjének magas logikai szintre állítása. *)
	CELL_ALL_Stop_Bit[0] := TRUE;
	CELL_ALL_Stop_Bit[1] := TRUE;
	CELL_ALL_Stop_Bit[2] := TRUE;

(* Mintavételezés eredményének feldolgozása, ha a vész-stop nem lett megnyomva. *)
ELSE
	CV_Robots_Update_Needed := FALSE;
	CV_Robots_Up_To_Date := FALSE;
	CV_Acknowledge_Needed := FALSE;

	(* A robotkonfigurációk módosítása, ha a mintavételezés eredménye alapján az operátor a rácson kívül tartózkodik és az utolsó ismert pozíciója ettől eltér. *)
	IF SAFETY_Logical_LOW > 0 AND SAFETY_Logical_HIGH = 0 AND SAFETY_Operator_Position <> 1 THEN
		(* Az új pozíció beálítása és a frissítés megkövetelése. *)
		SAFETY_Operator_Position := 1;
		CV_Robots_Update_Needed := TRUE;
		
		(* Az 1-es cella robotjainak felgyorsítása. *)
		CELL_ALL_Stop_Bit[0] := FALSE;
		CELL_ALL_Speed_Bit[0] := TRUE;
		
		(* A 2-es cella robotjainak felgyorsítása. *)
		CELL_ALL_Stop_Bit[1] := FALSE;
		CELL_ALL_Speed_Bit[1] := TRUE;
		
		(* A 3-as cella érintetlenül hagyása. *)
		CELL_ALL_Stop_Bit[2] := FALSE;
		CELL_ALL_Speed_Bit[2] := TRUE;
	
	(* A robotkonfigurációk módosítása, ha a mintavételezés eredménye alapján az operátor szemrevételez és az utolsó ismert pozíciója ettől eltér. *)
	ELSIF SAFETY_Logical_LOW > 0 AND SAFETY_Logical_HIGH > 0 AND SAFETY_Operator_Position <> 2 THEN
		(* Az új pozíció beálítása és a frissítés megkövetelése. *)
		SAFETY_Operator_Position := 2;
		CV_Robots_Update_Needed := TRUE;
		
		(* Az 1-es cella robotjainak felgyorsítása. *)
		CELL_ALL_Stop_Bit[0] := FALSE;
		CELL_ALL_Speed_Bit[0] := TRUE;
		
		(* A 2-es cella robotjainak lelassítása. *)
		CELL_ALL_Stop_Bit[1] := FALSE;
		CELL_ALL_Speed_Bit[1] := FALSE;
		
		(* A 3-as cella érintetlenül hagyása. *)
		CELL_ALL_Stop_Bit[2] := FALSE;
		CELL_ALL_Speed_Bit[2] := TRUE;
		
	(* A robotkonfigurációk módosítása, ha a mintavételezés eredménye alapján az operátor javít és az utolsó ismert pozíciója ettől eltér. *)
	ELSIF SAFETY_Logical_LOW = 0 AND SAFETY_Logical_HIGH > 0 AND SAFETY_Operator_Position <> 3 THEN
		(* Az új pozíció beálítása és a frissítés illetve a nyugtázás megkövetelése. *)
		SAFETY_Operator_Position := 3;
		CV_Robots_Update_Needed := TRUE;
		CV_Acknowledge_Needed := TRUE;

		(* Az 1-es cella robotjainak lelassítása. *)
		CELL_ALL_Stop_Bit[0] := FALSE;
		CELL_ALL_Speed_Bit[0] := FALSE;
		
		(* A 2-es cella robotjainak megállítása. *)
		CELL_ALL_Stop_Bit[1] := TRUE;
		CELL_ALL_Speed_Bit[1] := FALSE;
		
		(* A 3-as cella érintetlenül hagyása. *)
		CELL_ALL_Stop_Bit[2] := FALSE;
		CELL_ALL_Speed_Bit[2] := TRUE;
	
	(* A módosítások mellózése, ha a mintavételezés eredménye alapján nem történt változás. *)
	ELSE
		(* A frissítés mellózésének beállítása. *)
		CV_Robots_Up_To_Date := TRUE;

	END_IF;
	
END_IF;

### Action SAFETY_Wait_For_Acknowledge

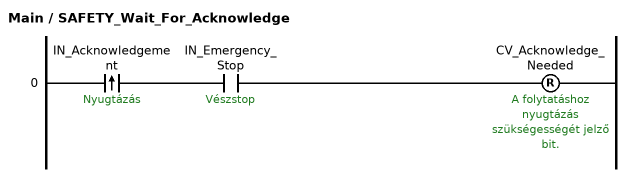
; rung 0
@LD IN_Acknowledgement  ; Nyugtázás
AND IN_Emergency_Stop  ; Vészstop
RSET CV_Acknowledge_Needed  ; A folytatáshoz nyugtázás szükségességét jelző bit.

### Action RESET_Wait_For_Startup

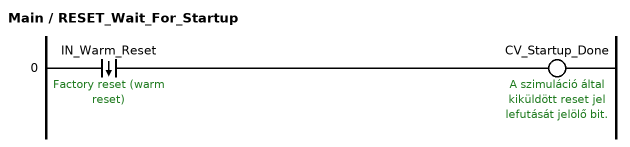
; rung 0
%LD IN_Warm_Reset  ; Factory reset (warm reset)
OUT CV_Startup_Done  ; A szimuláció által kiküldött reset jel lefutását jelölő bit.

### Action RESET_Wait_For_Reset

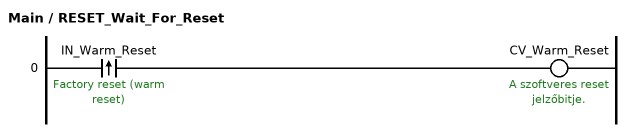
; rung 0
@LD IN_Warm_Reset  ; Factory reset (warm reset)
OUT CV_Warm_Reset  ; A szoftveres reset jelzőbitje.

### Subchart Robot_1_2_Operation
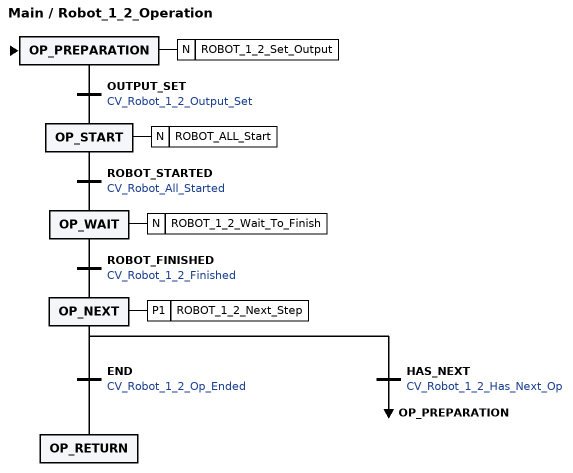
SUBCHART Robot_1_2_Operation:
ENTRY_STEP OP_PREPARATION :
ROBOT_1_2_Set_Output(N) ;
END_STEP
TRANSITION OUTPUT_SET FROM OP_PREPARATION TO OP_START
 := CV_Robot_1_2_Output_Set;
END_TRANSITION
STEP OP_START :
ROBOT_ALL_Start(N) ;
END_STEP
TRANSITION ROBOT_STARTED FROM OP_START TO OP_WAIT
 := CV_Robot_All_Started;
END_TRANSITION
STEP OP_WAIT :
ROBOT_1_2_Wait_To_Finish(N) ;
END_STEP
TRANSITION ROBOT_FINISHED FROM OP_WAIT TO OP_NEXT
 := CV_Robot_1_2_Finished;
END_TRANSITION
STEP OP_NEXT :
ROBOT_1_2_Next_Step(P1) ;
END_STEP
TRANSITION END (PRIORITY := 1) FROM OP_NEXT TO OP_RETURN
 := CV_Robot_1_2_Op_Ended;
END_TRANSITION
TRANSITION HAS_NEXT (PRIORITY := 2) FROM OP_NEXT TO OP_PREPARATION
 := CV_Robot_1_2_Has_Next_Op;
END_TRANSITION
RETURN_STEP OP_RETURN :
END_STEP
END_SUBCHART

### Subchart Robot_3_Operation
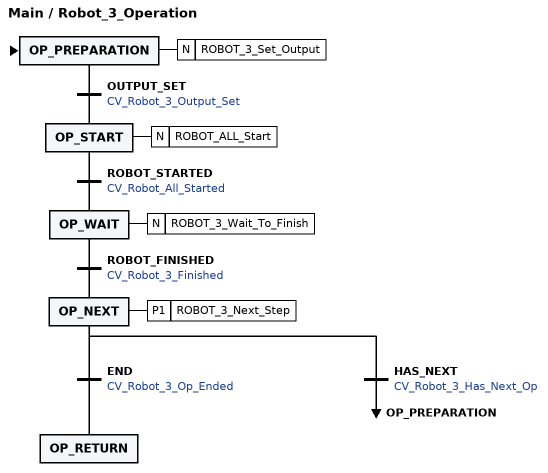
SUBCHART Robot_3_Operation:
ENTRY_STEP OP_PREPARATION :
ROBOT_3_Set_Output(N) ;
END_STEP
TRANSITION OUTPUT_SET FROM OP_PREPARATION TO OP_START
 := CV_Robot_3_Output_Set;
END_TRANSITION
STEP OP_START :
ROBOT_ALL_Start(N) ;
END_STEP
TRANSITION ROBOT_STARTED FROM OP_START TO OP_WAIT
 := CV_Robot_All_Started;
END_TRANSITION
STEP OP_WAIT :
ROBOT_3_Wait_To_Finish(N) ;
END_STEP
TRANSITION ROBOT_FINISHED FROM OP_WAIT TO OP_NEXT
 := CV_Robot_3_Finished;
END_TRANSITION
STEP OP_NEXT :
ROBOT_3_Next_Step(P1) ;
END_STEP
TRANSITION END (PRIORITY := 1) FROM OP_NEXT TO OP_RETURN
 := CV_Robot_3_Op_Ended;
END_TRANSITION
TRANSITION HAS_NEXT (PRIORITY := 2) FROM OP_NEXT TO OP_PREPARATION
 := CV_Robot_3_Has_Next_Op;
END_TRANSITION
RETURN_STEP OP_RETURN :
END_STEP
END_SUBCHART

### Subchart Crane_Operation
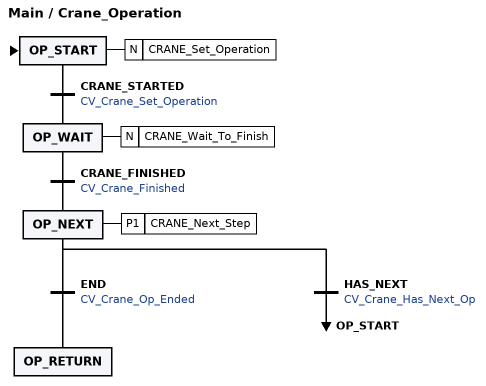
SUBCHART Crane_Operation:
ENTRY_STEP OP_START :
CRANE_Set_Operation(N) ;
END_STEP
TRANSITION CRANE_STARTED FROM OP_START TO OP_WAIT
 := CV_Crane_Set_Operation;
END_TRANSITION
STEP OP_WAIT :
CRANE_Wait_To_Finish(N) ;
END_STEP
TRANSITION CRANE_FINISHED FROM OP_WAIT TO OP_NEXT
 := CV_Crane_Finished;
END_TRANSITION
STEP OP_NEXT :
CRANE_Next_Step(P1) ;
END_STEP
TRANSITION END (PRIORITY := 1) FROM OP_NEXT TO OP_RETURN
 := CV_Crane_Op_Ended;
END_TRANSITION
TRANSITION HAS_NEXT (PRIORITY := 2) FROM OP_NEXT TO OP_START
 := CV_Crane_Has_Next_Op;
END_TRANSITION
RETURN_STEP OP_RETURN :
END_STEP
END_SUBCHART

### Subchart Safety_Get_Sample
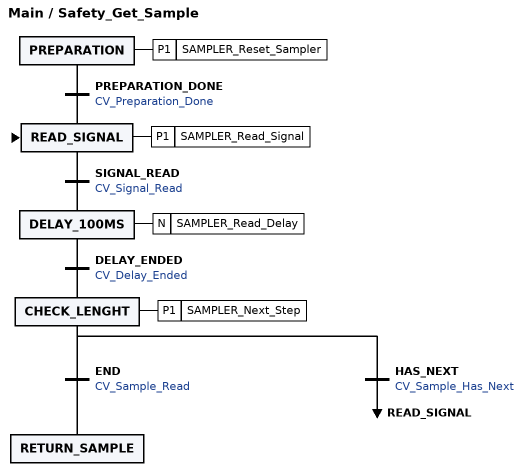
SUBCHART Safety_Get_Sample:
ENTRY_STEP PREPARATION :
SAMPLER_Reset_Sampler(P1) ;
END_STEP
TRANSITION SIGNAL_READ FROM READ_SIGNAL TO DELAY_100MS
 := CV_Signal_Read;
END_TRANSITION
STEP CHECK_LENGHT :
SAMPLER_Next_Step(P1) ;
END_STEP
TRANSITION END (PRIORITY := 1) FROM CHECK_LENGHT TO RETURN_SAMPLE
 := CV_Sample_Read;
END_TRANSITION
TRANSITION HAS_NEXT (PRIORITY := 2) FROM CHECK_LENGHT TO READ_SIGNAL
 := CV_Sample_Has_Next;
END_TRANSITION
RETURN_STEP RETURN_SAMPLE :
END_STEP
STEP DELAY_100MS :
SAMPLER_Read_Delay(N) ;
END_STEP
TRANSITION DELAY_ENDED FROM DELAY_100MS TO CHECK_LENGHT
 := CV_Delay_Ended;
END_TRANSITION
TRANSITION PREPARATION_DONE FROM PREPARATION TO READ_SIGNAL
 := CV_Preparation_Done;
END_TRANSITION
STEP READ_SIGNAL :
SAMPLER_Read_Signal(P1) ;
END_STEP
END_SUBCHART

### Subchart Update_Robots
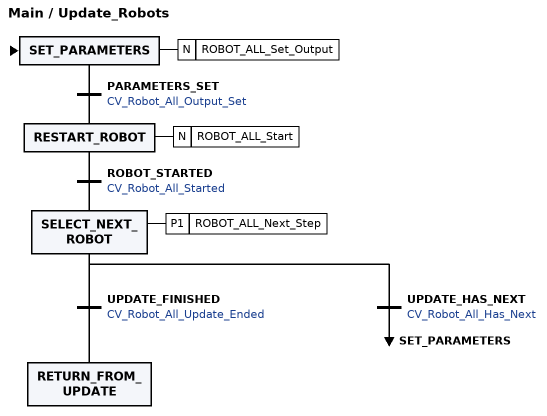
SUBCHART Update_Robots:
ENTRY_STEP SET_PARAMETERS :
ROBOT_ALL_Set_Output(N) ;
END_STEP
TRANSITION PARAMETERS_SET FROM SET_PARAMETERS TO RESTART_ROBOT
 := CV_Robot_All_Output_Set;
END_TRANSITION
STEP RESTART_ROBOT :
ROBOT_ALL_Start(N) ;
END_STEP
TRANSITION ROBOT_STARTED FROM RESTART_ROBOT TO SELECT_NEXT_ROBOT
 := CV_Robot_All_Started;
END_TRANSITION
STEP SELECT_NEXT_ROBOT :
ROBOT_ALL_Next_Step(P1) ;
END_STEP
TRANSITION UPDATE_FINISHED (PRIORITY := 1) FROM SELECT_NEXT_ROBOT TO RETURN_FROM_UPDATE
 := CV_Robot_All_Update_Ended;
END_TRANSITION
TRANSITION UPDATE_HAS_NEXT (PRIORITY := 2) FROM SELECT_NEXT_ROBOT TO SET_PARAMETERS
 := CV_Robot_All_Has_Next;
END_TRANSITION
RETURN_STEP RETURN_FROM_UPDATE :
END_STEP
END_SUBCHART